INTERFACE ITF_MCHMIPrepareScreen_00_03_Init

METHOD PUBLIC LinkDataHMI_00_03 : BOOL
VAR_INPUT
	refstData				: REFERENCE TO ST_MCHMIPrepareScreen_00_03;
END_VAR
END_METHOD

END_INTERFACE

(* stored: Version 1.1.0.1
   Itf ITF_MCHMIPrepareScreen_00_03_Init: Id {a67cc089-2353-0aba-0315-e080814fc2be}
   Method LinkDataHMI_00_03: Id {a070e933-41e0-0a60-07c2-cf6188eb3af4} *)
